// A -=B
FUNCTION vecSelfSub : BOOL
VAR_IN_OUT
	vecA :ARRAY[*] OF LREAL;
END_VAR

VAR_IN_OUT CONSTANT
	vecB :ARRAY[*] OF LREAL;
END_VAR

VAR
	m,i :DINT;
 
END_VAR

m:=UPPER_BOUND(vecA,1);

FOR i:=1 TO m DO
		vecA[i]:=vecA[i]-vecB[i];
END_FOR

END_FUNCTION

(* stored: Version 1.1.0.1, ProductVersion 3.1.4024.11
   POU vecSelfSub: Id {ef64eff1-9176-463b-b3b0-4b2081ef4cad}, SpecialFunc None *)
